{attribute 'TcEncoding':='UTF-8'}
TYPE Utf8String : T_MaxString; END_TYPE

(* stored: Version 1.1.0.1
   DUT Utf8String: Id {81066540-0754-0f38-109d-b7019ca0b434} *)
